
FUNCTION CB_div_t_dint : TIME


TITLE = ' Dividing a time '
VERSION : '1.0'
AUTHOR  : CB
NAME    : divTiDi
FAMILY  : TNI

VAR_INPUT
    IN0 : TIME;
    IN1 : DINT;
END_VAR

BEGIN
    CB_div_t_dint := IN0 / IN1;
END_FUNCTION
